TYPE E_HMI_DriveStatus :
(
	E_DRIVE_UNKNOWN := 0,
	E_DRIVE_SPOPPED := 1,
	E_DRIVE_RUNING := 2,
	E_DRIVE_ERROR := 3
);
END_TYPE

(* stored: Version 1.1.0.1
   DUT E_HMI_DriveStatus: Id {30a76562-a2f9-4391-ad18-830ee7c84e54} *)
